{attribute 'pack_mode' := '2'}
TYPE ST_MOVER_CTRL :
STRUCT
  Cmd             : E_MOVER_CTRL;  // order to execute on mover
END_STRUCT
END_TYPE

(* stored: Version 1.1.0.1
   DUT ST_MOVER_CTRL: Id {4817b66c-008d-4e7b-9e8c-18fdcbd7fa0d} *)
